(* PLC project MotionTest1, Higen MCL 1 *)
(* stored: creationDateTime 2012-01-06T15:20:13, modificationDateTime 2026-03-16T00:08:53 *)

PROGRAM main
  VAR
    clock : ULINT;
    Done : BOOL;
    Axis : AXIS_REF;
    switch : MC_Power;
    readpos : MC_ReadActualPosition;
    Pn : LREAL;
    Vn : LREAL;
    setpos : MC_SetPosition;
    readspeed : MC_ReadParameter;
    my_simulated_axis : MC_Sim;
    speeed : MC_MoveVelocity;
  END_VAR

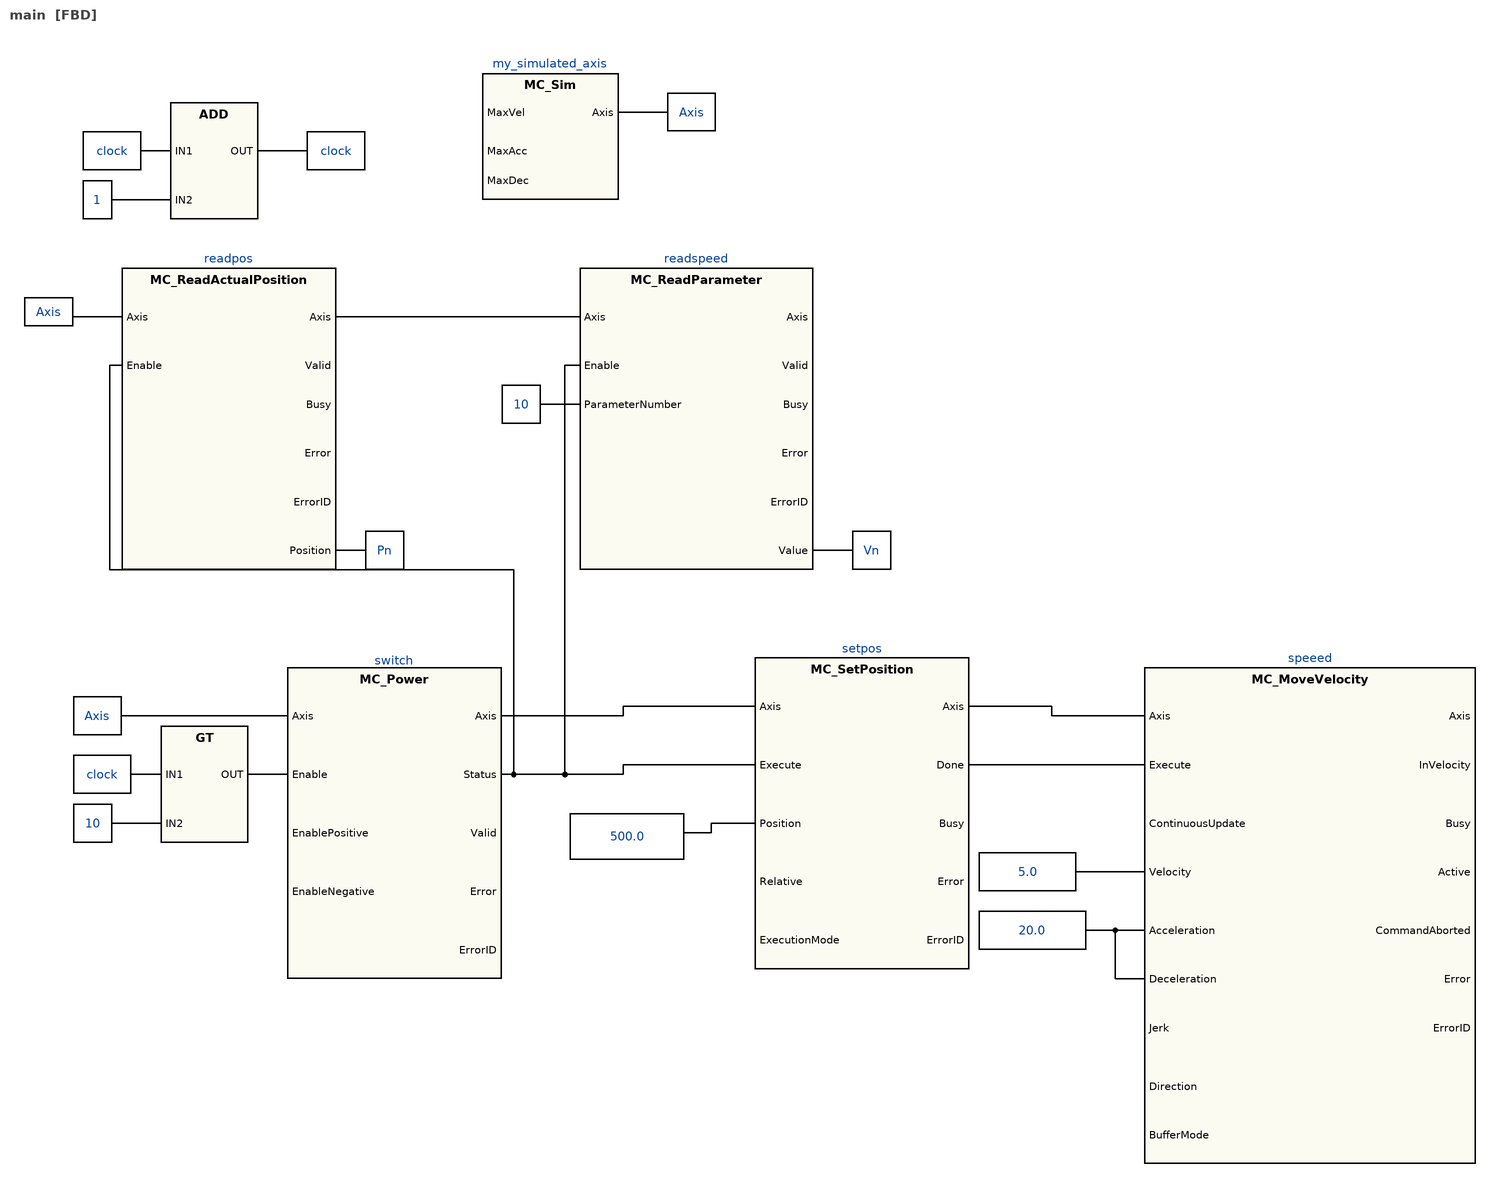
(* FBD diagram, written out as Structured Text *)
clock := clock + 1;
switch(Axis := Axis, Enable := clock > 10);
readpos(Axis := Axis, Enable := switch.Status);
Pn := readpos.Position;
readspeed(Axis := readpos.Axis, Enable := switch.Status, ParameterNumber := 10);
Vn := readspeed.Value;
my_simulated_axis();
Axis := my_simulated_axis.Axis;
setpos(Axis := switch.Axis, Execute := switch.Status, Position := 500.0);
speeed(Axis := setpos.Axis, Execute := setpos.Done, Velocity := 5.0, Acceleration := 20.0, Deceleration := 20.0);
END_PROGRAM

CONFIGURATION conf
  RESOURCE res ON PLC
    TASK milisecond(INTERVAL := T#1ms, PRIORITY := 0);
    PROGRAM maininstance WITH milisecond : main;
  END_RESOURCE
END_CONFIGURATION
